(* Schneider Machine Expert - Basic project plc-coaster, file version 3.0.0.0 *)
(* ProjectInformations: Name=New project *)

HARDWARE
  Cpu 0: TM221CE16R
  EthernetConfiguration: NetworkName=M221, IpAllocationMode=FixedAddress, IpAddress=0.0.0.0, SubnetMask=0.0.0.0
  SerialLineConfiguration: Baud=Baud19200, Parity=ParityEven, DataBits=DataBits8, StopBits=StopBits1, PhysicalMedium=PhysicalMediumRs485, TransmissionMode=TransmissionModeModbusRtu, SlaveId=1, Addressing=SlaveAddressing
  MastTask: UsePeriodScanMode=false, PeriodScan=100
  FastTask: Period=255
  CpuBehavior: StartingMode=StartAsPreviousState, AutoSaveRamOnEeprom=true, WatchdogPeriod=250

SYMBOLS  (address, symbol, comment, settings)
  %M0       ALL_RESTRAINTS_OK
  %M1       FAULT_LATCH
  %I0.0     RESTRAINT_ROW1
  %I0.1     RESTRAINT_ROW2
  %I0.2     RESTRAINT_ROW3
  %I0.3     READY_PB
  %I0.4     ESTOP
  %I0.5     GATE_CLOSED
  %I0.6     FAULT_RESET_PB
  %Q0.0     DISPATCH_PERMISSIVE
  %Q0.1     BRAKE_RELEASE
  %Q0.2     FAULT_LAMP

POU New POU
  (* SectionNumber=1 *)

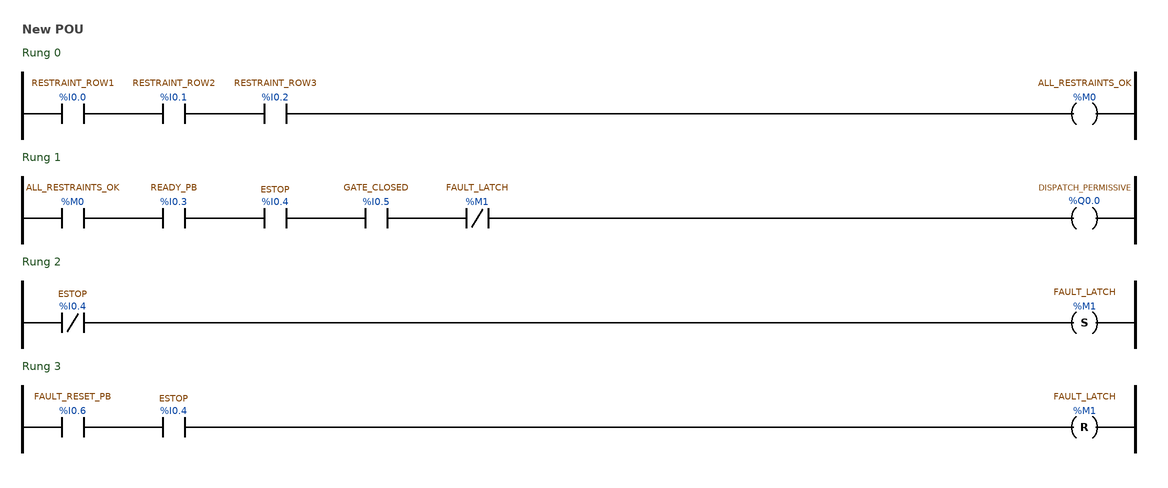

// Rung 0
  LD %I0.0                (* RESTRAINT_ROW1 *)
  AND %I0.1               (* RESTRAINT_ROW2 *)
  AND %I0.2               (* RESTRAINT_ROW3 *)
  ST %M0                  (* ALL_RESTRAINTS_OK *)
  // as ST:
  //   ALL_RESTRAINTS_OK := RESTRAINT_ROW1 AND RESTRAINT_ROW2 AND RESTRAINT_ROW3;

// Rung 1
  LD %M0                  (* ALL_RESTRAINTS_OK *)
  AND %I0.3               (* READY_PB *)
  AND %I0.4               (* ESTOP *)
  AND %I0.5               (* GATE_CLOSED *)
  ANDN %M1                (* FAULT_LATCH *)
  ST %Q0.0                (* DISPATCH_PERMISSIVE *)
  // as ST:
  //   DISPATCH_PERMISSIVE := ALL_RESTRAINTS_OK AND READY_PB AND ESTOP AND GATE_CLOSED AND NOT FAULT_LATCH;

// Rung 2
  LDN %I0.4               (* ESTOP *)
  S %M1                   (* FAULT_LATCH *)
  // as ST:
  //   IF NOT ESTOP THEN FAULT_LATCH := TRUE; END_IF;

// Rung 3
  LD %I0.6                (* FAULT_RESET_PB *)
  AND %I0.4               (* ESTOP *)
  R %M1                   (* FAULT_LATCH *)
  // as ST:
  //   IF FAULT_RESET_PB AND ESTOP THEN FAULT_LATCH := FALSE; END_IF;
